% RSLogix 500 project T_RTO.RSS, saved by version 8.30.00.16 %
PROJECT "UNTITLED"    % processor: Bul.1763 MicroLogix 1100 Series B %

PROGRAM FILES
  LAD 2   6 rungs

DATA FILES
  O0 OUTPUT  4 elements
  I1 INPUT  6 elements
  S2 STATUS  66 elements
  B3 BINARY  1 elements
  T4 TIMER  1 elements
  C5 COUNTER  1 elements
  R6 CONTROL  1 elements
  N7 INTEGER  1 elements
  F8 FLOAT  1 elements

LADDER 2
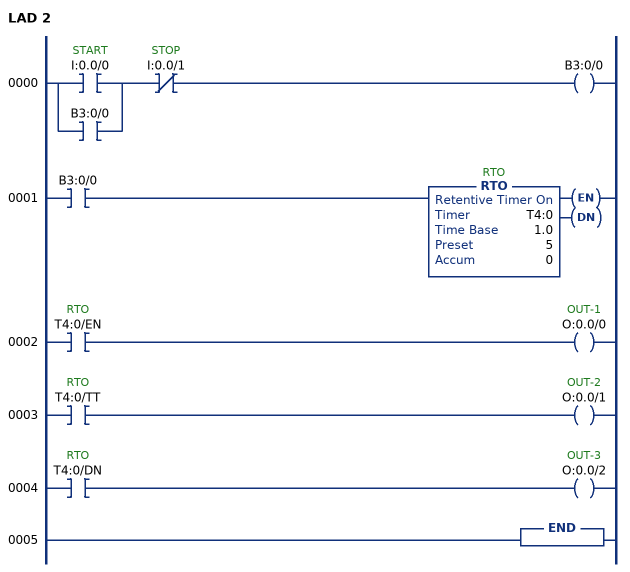
% Rung: 0 %
SOR BST XIC I:0.0/0 NXB XIC B3:0/0 BND XIO I:0.0/1 OTE B3:0/0 EOR
%   I:0.0/0  "START" %
%   I:0.0/1  "STOP" %
% Rung: 1 %
SOR XIC B3:0/0 RTO T4:0 1.0 5 0 EOR
%   T4:0  "RTO" %
% Rung: 2 %
SOR XIC T4:0/EN OTE O:0.0/0 EOR
%   T4:0  "RTO" %
%   O:0.0/0  "OUT-1" %
% Rung: 3 %
SOR XIC T4:0/TT OTE O:0.0/1 EOR
%   T4:0  "RTO" %
%   O:0.0/1  "OUT-2" %
% Rung: 4 %
SOR XIC T4:0/DN OTE O:0.0/2 EOR
%   T4:0  "RTO" %
%   O:0.0/2  "OUT-3" %
% Rung: 5 %
SOR END EOR

DATA TABLE (non-zero values as saved)
DATA T4
% .PRE .ACC %
% T4:0 % 5 0
